// TIA Portal V20 export
TYPE "NDD_Interlock_Horquilla"
   STRUCT
      PosHorq_Bloqueo : Bool;   // La Horquilla esta en Bloqueo para ir a la Posicion IN (Hacia el Elevador)
      MovHorq_Bloqueada : Bool;
      OrdenDeSalida : Bool;   // Orden de la Salida de la Paleta de la Horquilla
      FinOrdenDeSalida : Bool;
      DejarCarga_EntradaHorq : Bool;
      DejadaCarga_EntradaHorq : Bool;   // Aviso de Dejar la Paleta en la Horquilla
      RecogerCarga_SalidaHorq : Bool;   // Aviso de Recoger la Paleta de la Horquilla
      RecogidaCarga_SalidaHorq : Bool;
      AVTF_EntradaHorq : Bool;   // Aviso de Entrada de la Paleta en la Horquilla
      PTF_EntradaHorq : Bool;   // Permiso de Entrada de la Paleta en la Horquilla
      FTF_EntradaHorq : Bool;   // Fin de la Entrada de la Paleta en la Horquilla
      AVTF_SalidaHorq : Bool;   // Aviso de Salida de la Paleta en la Horquilla
      PTF_SalidaHorq : Bool;   // Permiso de Salida de la Paleta en la Hoquilla
      FTF_SalidaHorq : Bool;   // Fin de la Salida de la Paleta en la Hoprquilla
      Libre_16 : Bool;
      DesHabilitarBarrera_Down : Bool;
      ConCarga_Horq : Bool;
      Horq_Out : Bool;
      Horq_In : Bool;
      Horq_SeguridadUp : Bool;
      Horq_SeguridadDown : Bool;
      Libre_25 : Bool;
      Libre_26 : Bool;
      Horq_EnReset : Bool;
      Horq_EnCarga : Bool;
      Horq_EnVacio : Bool;
      Horq_Entrando : Bool;
      Horq_Saliendo : Bool;
      Libre_35 : Bool;
      Libre_36 : Bool;
      Libre_37 : Bool;
   END_STRUCT;
END_TYPE
